TYPE ST_Ampel_Steuerung :
STRUCT
	Freigabe			: ST_Steuerung_auto_manu_BOOL;
	Quittierung			: BOOL;
END_STRUCT
END_TYPE

(* stored: Version 1.1.0.1, ProductVersion 3.1.4024.9
   DUT ST_Ampel_Steuerung: Id {e28a3a3e-5893-4097-9afb-e5124ba340e3} *)
